INTERFACE I_PUMP_WITH_BYPASS EXTENDS I_ENGINE

METHOD M_Bypass : BOOL
VAR_INPUT
  bEnable:        BOOL;
END_VAR
END_METHOD

PROPERTY P_BypassState : BOOL
GET
END_GET
END_PROPERTY

END_INTERFACE

(* stored: Version 1.1.0.1, ProductVersion 3.1.4024.12
   Itf I_PUMP_WITH_BYPASS: Id {87bb4e59-4d3d-4eca-9708-e001aa95480a}
   Method M_Bypass: Id {72b254d6-ba26-4dd7-9fb7-0c2af2a167d6}
   Property P_BypassState: Id {c60fc096-cb52-4851-91da-72a141552ee4}
   Get Get: Id {f1d3a4af-0061-4814-b5bf-62d2d9a3dde7} *)
